{attribute 'linkalways'} 
{attribute 'no_explicit_call' := 'This FB is a CLASS and must be accessed using methods or properties'}
{attribute 'enable_dynamic_creation'}
FUNCTION_BLOCK ABSTRACT UserDefinedDatatypeBase EXTENDS DatatypeBase IMPLEMENTS I_UserDefinedDatatype
VAR
END_VAR

PROPERTY PUBLIC ABSTRACT Identifier : T_MAXSTRING
GET
END_GET
END_PROPERTY

METHOD PROTECTED OnSerializeTypeWith
VAR_INPUT
	Serializer : I_Serializer;
END_VAR
SUPER^.OnSerializeTypeWith(Serializer);
Serializer.AddKeyString('identifier',Identifier);
END_METHOD

END_FUNCTION_BLOCK

(* stored: Version 1.1.0.1, ProductVersion 3.1.4024.12
   POU UserDefinedDatatypeBase: Id {46f1ce56-9ece-0468-3f0b-6f6310f7daa4}, SpecialFunc None
   Folder Protected: Id {c0485087-525e-03d0-0c3e-1ead28aca980}
   Property Identifier: Id {fad1b093-141e-0c94-3cbf-d2814230ee8f}
   Get Get: Id {0ba07a67-9506-0b52-2c39-54987f0097d7}
   Method OnSerializeTypeWith: Id {e57435fa-f18e-0790-33a1-e7b24c80ba5a} *)
